RESOURCE_TYPE _WaterHeaterPlantAndController
  (* Standard: 61499-2 *)
  (* Version 0.1, 2017-00-01, hpea485, UOA *)
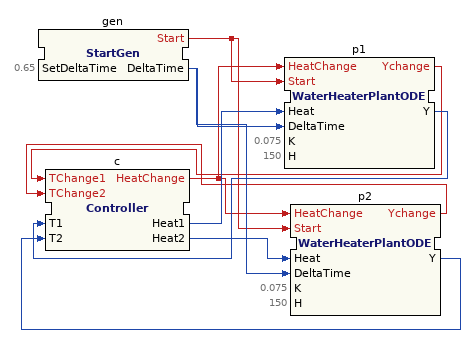
  FBS
    p1 : WaterHeaterPlantODE(K := 0.075, H := 150);
    p2 : WaterHeaterPlantODE(K := 0.075, H := 150);
    c : Controller;
    gen : StartGen(SetDeltaTime := 0.65);
  END_FBS
  EVENT_CONNECTIONS
    p1.Ychange TO c.TChange1;
    p2.Ychange TO c.TChange2;
    c.HeatChange TO p1.HeatChange;
    c.HeatChange TO p2.HeatChange;
    gen.Start TO p1.Start;
    gen.Start TO p2.Start;
  END_CONNECTIONS
  DATA_CONNECTIONS
    p1.Y TO c.T1;
    p2.Y TO c.T2;
    c.Heat1 TO p1.Heat;
    c.Heat2 TO p2.Heat;
    gen.DeltaTime TO p1.DeltaTime;
    gen.DeltaTime TO p2.DeltaTime;
  END_CONNECTIONS
END_RESOURCE_TYPE
